TYPE ST_HeatPump_Get :
STRUCT
	HeatPumpState 	: 	eHeatPumpState;
	Setpoint		:	REAL;
	Events			: 	ST_HeatPumpEvents;
	
	HeatpumpData	:	ST_HeatpumpData;
END_STRUCT
END_TYPE

(* stored: Version 1.1.0.1, ProductVersion 3.1.4026.18
   DUT ST_HeatPump_Get: Id {432044be-355d-481a-bff6-9f48e6ab4142} *)
